FUNCTION_BLOCK EM_Gantry
VAR_INPUT
END_VAR
VAR_OUTPUT
END_VAR
VAR
END_VAR

// NETWORK 1

END_FUNCTION_BLOCK

(* stored: Version 1.1.0.1, ProductVersion 3.1.4024.13
   POU EM_Gantry: Id {7ef900b8-5b82-429c-a2bf-4415c503f2ac}, SpecialFunc None *)
